{attribute 'qualified_only'}
VAR_GLOBAL PERSISTENT

    // Kompanzasyon grupları konfigürasyonu
    astCompensationGroups : ARRAY[0..GVL_CompensationGroup.MAX_COMPENSATION_GROUPS-1] OF ST_CompensationGroup;  // Tüm grupların kondansatör bilgileri
    nConfiguredGroups : INT;                                                                                    // Toplam konfigüre edilmiş grup sayısı
    
    // Grup aktif durumları
    abGroupActive : ARRAY[0..GVL_CompensationGroup.MAX_COMPENSATION_GROUPS-1] OF BOOL;                         // Her grubun aktif/pasif durumu
    
    // Ana kesici HMI bilgileri
    stMainDisconnectorHMI : ST_DisconnectorHMI;                                                               // Ana kesici durum ve kontrol bilgileri
    
    // Grup 1 Kontaktör HMI bilgileri
    stGroup1_ContactorHMI : ST_ContactorHMI;                                                                   // Grup 1 kontaktör durum ve kontrol bilgileri
    
    // Grup 2 Kontaktör HMI bilgileri
    stGroup2_ContactorHMI : ST_ContactorHMI;                                                                   // Grup 2 kontaktör durum ve kontrol bilgileri
    
    // Grup 3 Kontaktör HMI bilgileri
    stGroup3_ContactorHMI : ST_ContactorHMI;                                                                   // Grup 3 kontaktör durum ve kontrol bilgileri
    
    // Grup 4 Kontaktör HMI bilgileri
    stGroup4_ContactorHMI : ST_ContactorHMI;                                                                   // Grup 4 kontaktör durum ve kontrol bilgileri
    
    // Grup 5 Kontaktör HMI bilgileri
    stGroup5_ContactorHMI : ST_ContactorHMI;                                                                   // Grup 5 kontaktör durum ve kontrol bilgileri
    
    // Grup 6 Kontaktör HMI bilgileri
    stGroup6_ContactorHMI : ST_ContactorHMI;                                                                   // Grup 6 kontaktör durum ve kontrol bilgileri
   
   // Grup 7 Kontaktör HMI bilgileri
   stGroup7_ContactorHMI : ST_ContactorHMI;                                                                   // Grup 7 kontaktör durum ve kontrol bilgileri
   
   // Grup 8 Kontaktör HMI bilgileri
   stGroup8_ContactorHMI : ST_ContactorHMI;                                                                   // Grup 8 kontaktör durum ve kontrol bilgileri
   
   // Grup 9 Kontaktör HMI bilgileri
   stGroup9_ContactorHMI : ST_ContactorHMI;                                                                   // Grup 9 kontaktör durum ve kontrol bilgileri
   
   // Grup 10 Kontaktör HMI bilgileri
   stGroup10_ContactorHMI : ST_ContactorHMI;                                                                  // Grup 10 kontaktör durum ve kontrol bilgileri
END_VAR

(* stored: Version 1.1.0.1, ProductVersion 3.1.4024.15
   GVL GVL_LVCP1: Id {1effb160-27c6-4b6d-b40b-6a4dc74e0876} *)
